TYPE E_MoMa_1stHierarchy_States :
(
	Init,
	IdleState,
	UserInteraction, 
	Prepare,
	Implementation,
	Clear,
	ServiceNeeded
)UDINT;
END_TYPE

(* stored: Version 1.1.0.1, ProductVersion 3.1.4024.11
   DUT E_MoMa_1stHierarchy_States: Id {10ce00cc-d7fa-4567-a974-ec2e7a693170} *)
